ABB RobotStudio station: socketTest.rspag

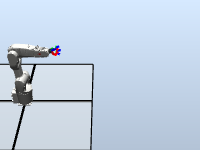
--- station ---
Station Station (saved by RobotStudio 6.7.7936.1011)
Controller pcsdk
  mechanical unit ROB_1: IRB1200_5_90_STD_02, 6 joints, base frame (0, 0, 0) mm
Layout (positions relative to the parent item):
  - IRB1200_5_90_STD_02 [mechanism, from Robots\IRB1200_5_90_STD_02.rslib] at (0, 0, 0) mm; joint values [-0.1777, -0.1118, 0.0853, -0.0088, -0.4461, 0.0081] (rad or m)
Targets, tools, work objects and paths stored in the station and not in the controller backup, written as RAPID:
! task T_ROB1
MODULE Module1
  VAR robtarget pTarget:=[[0,0,0],[1,0,0,0],[0,0,0,0],[9E+09,9E+09,9E+09,9E+09,9E+09,9E+09]];
  VAR jointtarget jTarget:=[[0,0,0,0,0,0],[9E+09,9E+09,9E+09,9E+09,9E+09,9E+09]];
  CONST jointtarget joint1:=[[0,0,0,0,30,0],[9E+09,9E+09,9E+09,9E+09,9E+09,9E+09]];
  CONST jointtarget joint2:=[[0,0,0,0,-30,0],[9E+09,9E+09,9E+09,9E+09,9E+09,9E+09]];
ENDMODULE


--- Backups/pcsdk/RAPID/TASK1/PROGMOD/Module1.mod ---
MODULE Module1
    var robtarget pTarget;
    VAR jointtarget jTarget;

    PROC main()
        !Add your code here
        TPWrite"Hello";
    ENDPROC

    PROC MoveLinear()
        MoveL pTarget,v1000,fine,tool0;
    ENDPROC

    PROC moveJoint()
        MoveAbsJ jTarget,v1000,fine,tool0;
    ENDPROC
ENDMODULE

--- Backups/pcsdk/SYSPAR/EIO.cfg ---
EIO:CFG_1.0:6:1::
#
INDUSTRIAL_NETWORK:

      -Name "DeviceNet" -Label "DeviceNet Master/Slave Network" -Address "2"
#
DEVICENET_DEVICE:

      -Name "d652"
#
DEVICENET_INTERNAL_DEVICE:

      -Name "DN_Internal_Device" -VendorName "ABB Robotics"\
      -ProductName "DeviceNet Internal Slave Device"
#
EIO_SIGNAL:

      -Name "do1" -SignalType "DO" -Device "d652" -DeviceMap "0" -Access "All"

      -Name "di1" -SignalType "DI" -Device "d652" -DeviceMap "0" -Access "All"
